// TwinCAT 3 PLC project work_flow_interface
// ProgramVersion: 3.1.4024.0
// libraries:
//   Tc2_Standard, * (Beckhoff Automation GmbH)
//   Tc2_System, * (Beckhoff Automation GmbH)
//   Tc3_Module, * (Beckhoff Automation GmbH)
// project tree:
//   / PlcTask.TcTTO
//   POUs/ FB_StringBuilder.TcPOU, I_StringBuilder.TcIO, MAIN.TcPOU
// (motion and I/O tree: see PLC project work flow reference)
// real-time tasks:
//   TASK PlcTask3: cycle T#10ms, priority 20, ADS port 350
//   TASK PlcTask1: cycle T#10ms, priority 21, ADS port 351
//   TASK PlcTask2: cycle T#10ms, priority 22, ADS port 352

CONFIGURATION work_flow_interface
    RESOURCE PLC ON TwinCAT3
        TASK PlcTask(INTERVAL := T#10ms, PRIORITY := 22);
        PROGRAM MAIN WITH PlcTask : MAIN;
    END_RESOURCE
END_CONFIGURATION

// ---- POUs/I_StringBuilder.TcIO
INTERFACE I_StringBuilder EXTENDS __SYSTEM.IQueryInterface

METHOD Append : I_StringBuilder
VAR_INPUT
	sText : STRING;
END_VAR
END_METHOD

METHOD Clear : I_StringBuilder
VAR_INPUT
END_VAR
END_METHOD

METHOD ToString : STRING
VAR_INPUT
END_VAR
END_METHOD

END_INTERFACE

// ---- POUs/MAIN.TcPOU
PROGRAM MAIN
VAR
	// print out 'Hello world'
	fbStringBuilder : FB_StringBuilder;
	iStringBuilder	: I_StringBuilder := fbStringBuilder;
	sResult1 : STRING;
	sResult2 : STRING;
	bTest : BOOL;
END_VAR

IF bTest THEN
	// Function Block Instance
	sResult1 := fbStringBuilder.Clear()
							.Append('H')
							.Append('e')
							.Append('l')
							.Append('l')
							.Append('o')
							.Append(' ')
							.Append('W')
							.Append('o')
							.Append('r')
							.Append('l')
							.Append('d')
							.ToString();
	// Interface 
	sResult2 := iStringBuilder.Clear()
							.Append('H')
							.Append('e')
							.Append('l')
							.Append('l')
							.Append('o')
							.Append(' ')
							.Append('W')
							.Append('o')
							.Append('r')
							.Append('l')
							.Append('d')
							.ToString();
	bTest := FALSE;
END_IF

END_PROGRAM

// ---- POUs/FB_StringBuilder.TcPOU
FUNCTION_BLOCK FB_StringBuilder IMPLEMENTS I_StringBuilder
VAR
	sContent : STRING; // Store temporary strings;
END_VAR

METHOD Append : I_StringBuilder
VAR_INPUT
	sText : STRING;
END_VAR
sContent := CONCAT(STR1 := sContent, STR2 := sText);
Append := THIS^;
END_METHOD

METHOD Clear : I_StringBuilder
VAR_INPUT
END_VAR
sContent := '';
Clear := THIS^;
END_METHOD

METHOD ToString : STRING
VAR_INPUT
END_VAR
ToString := sContent; // return internal content
END_METHOD

END_FUNCTION_BLOCK
